PROGRAM Vision_Calibration
VAR
	
	Always_ON					:	BOOL	:=TRUE;	//상시ON
	Always_OFF					:	BOOL	:=FALSE;//상시OFF
	
	GVL_Calibration_Step: BOOL;
	TON_0: TON;
	TON_1: TON;
	TON_2: TON;
END_VAR
VAR // added by the converter: edge detectors and wires of the graphical bodies
    _w1 : BOOL;
END_VAR

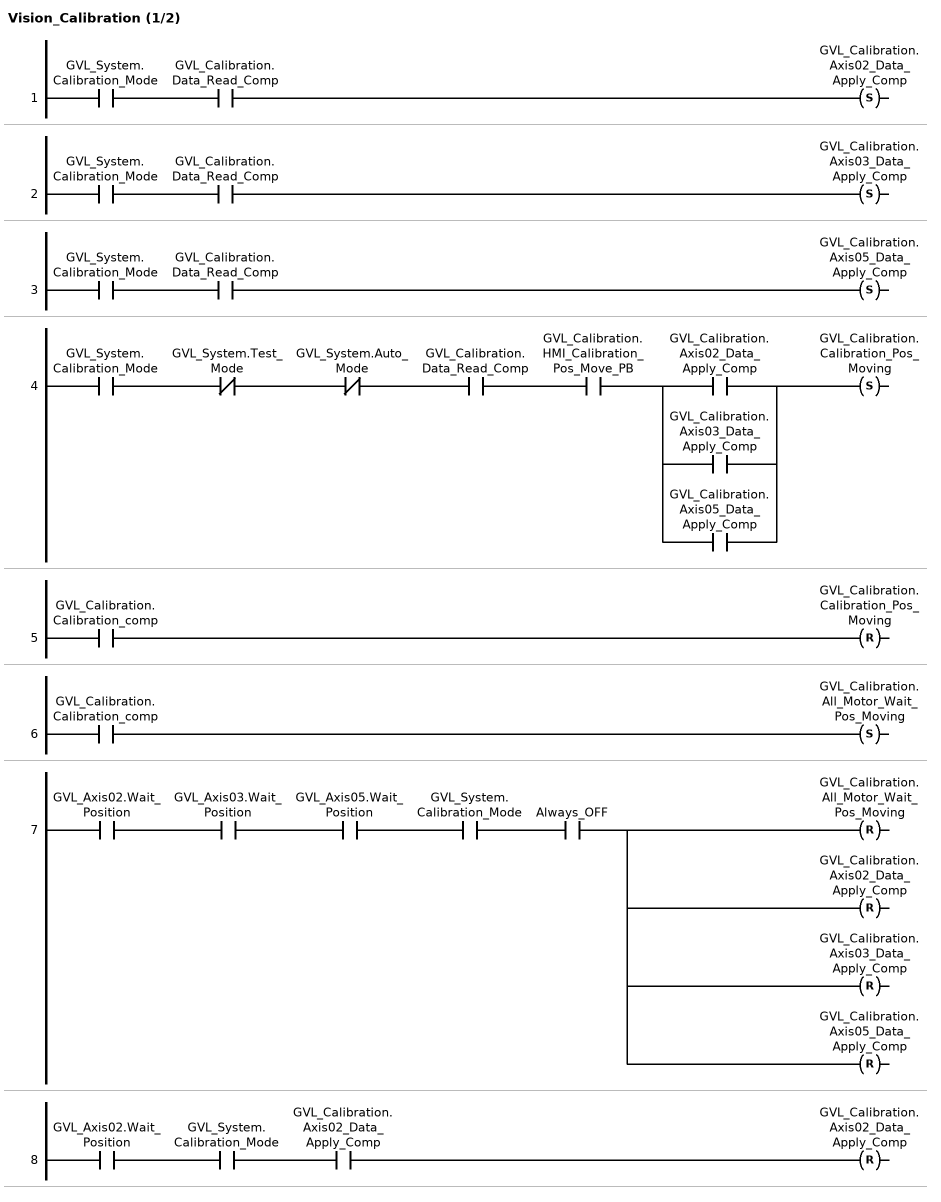
// NETWORK 1
GVL_Calibration.Axis02_Data_Apply_Comp S= GVL_System.Calibration_Mode AND GVL_Calibration.Data_Read_Comp;

// NETWORK 2
GVL_Calibration.Axis03_Data_Apply_Comp S= GVL_System.Calibration_Mode AND GVL_Calibration.Data_Read_Comp;

// NETWORK 3
GVL_Calibration.Axis05_Data_Apply_Comp S= GVL_System.Calibration_Mode AND GVL_Calibration.Data_Read_Comp;

// NETWORK 4
GVL_Calibration.Calibration_Pos_Moving S= GVL_System.Calibration_Mode AND NOT GVL_System.Test_Mode AND NOT GVL_System.Auto_Mode AND GVL_Calibration.Data_Read_Comp AND GVL_Calibration.HMI_Calibration_Pos_Move_PB AND (GVL_Calibration.Axis02_Data_Apply_Comp OR GVL_Calibration.Axis03_Data_Apply_Comp OR GVL_Calibration.Axis05_Data_Apply_Comp);

// NETWORK 5
GVL_Calibration.Calibration_Pos_Moving R= GVL_Calibration.Calibration_comp;

// NETWORK 6
GVL_Calibration.All_Motor_Wait_Pos_Moving S= GVL_Calibration.Calibration_comp;

// NETWORK 7
_w1 := GVL_Axis02.Wait_Position AND GVL_Axis03.Wait_Position AND GVL_Axis05.Wait_Position AND GVL_System.Calibration_Mode AND Always_OFF;
GVL_Calibration.All_Motor_Wait_Pos_Moving R= _w1;
GVL_Calibration.Axis02_Data_Apply_Comp R= _w1;
GVL_Calibration.Axis03_Data_Apply_Comp R= _w1;
GVL_Calibration.Axis05_Data_Apply_Comp R= _w1;

// NETWORK 8
GVL_Calibration.Axis02_Data_Apply_Comp R= GVL_Axis02.Wait_Position AND GVL_System.Calibration_Mode AND GVL_Calibration.Axis02_Data_Apply_Comp;

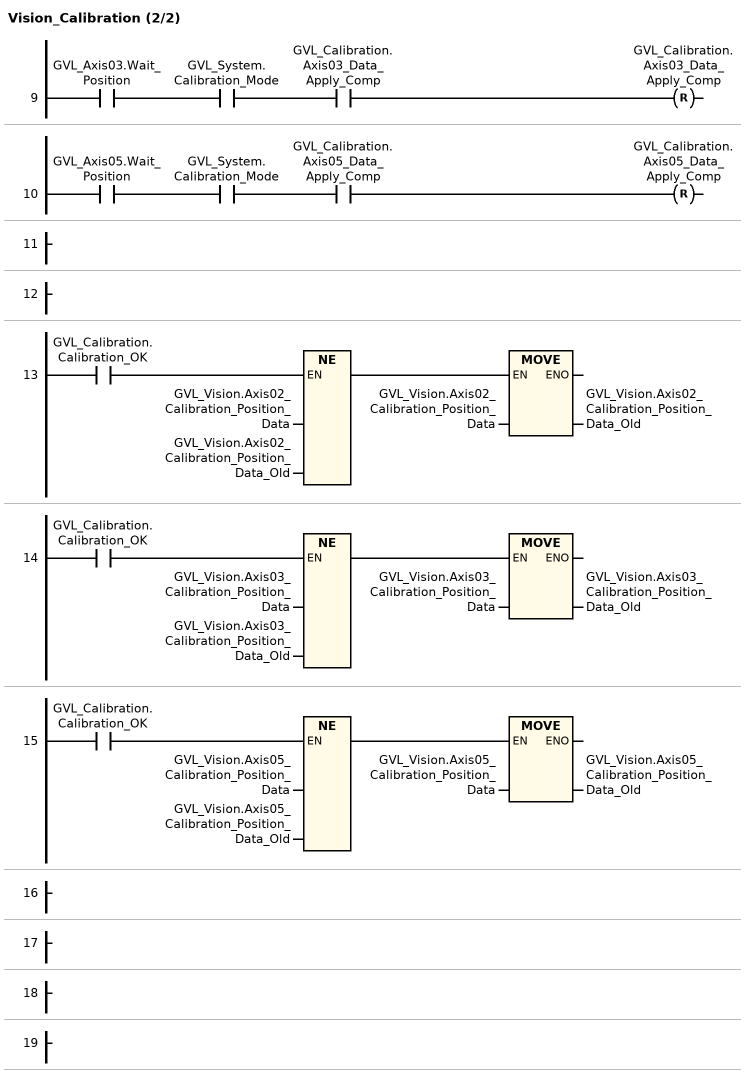
// NETWORK 9
GVL_Calibration.Axis03_Data_Apply_Comp R= GVL_Axis03.Wait_Position AND GVL_System.Calibration_Mode AND GVL_Calibration.Axis03_Data_Apply_Comp;

// NETWORK 10
GVL_Calibration.Axis05_Data_Apply_Comp R= GVL_Axis05.Wait_Position AND GVL_System.Calibration_Mode AND GVL_Calibration.Axis05_Data_Apply_Comp;

// NETWORK 11

// NETWORK 12

// NETWORK 13
IF GVL_Calibration.Calibration_OK AND GVL_Vision.Axis02_Calibration_Position_Data <> GVL_Vision.Axis02_Calibration_Position_Data_Old THEN
    GVL_Vision.Axis02_Calibration_Position_Data_Old := GVL_Vision.Axis02_Calibration_Position_Data;
END_IF

// NETWORK 14
IF GVL_Calibration.Calibration_OK AND GVL_Vision.Axis03_Calibration_Position_Data <> GVL_Vision.Axis03_Calibration_Position_Data_Old THEN
    GVL_Vision.Axis03_Calibration_Position_Data_Old := GVL_Vision.Axis03_Calibration_Position_Data;
END_IF

// NETWORK 15
IF GVL_Calibration.Calibration_OK AND GVL_Vision.Axis05_Calibration_Position_Data <> GVL_Vision.Axis05_Calibration_Position_Data_Old THEN
    GVL_Vision.Axis05_Calibration_Position_Data_Old := GVL_Vision.Axis05_Calibration_Position_Data;
END_IF

// NETWORK 16

// NETWORK 17

// NETWORK 18

// NETWORK 19

END_PROGRAM

(* stored: Version 1.1.0.1, ProductVersion 3.1.4024.15
   POU Vision_Calibration: Id {cb4ac576-599e-4820-9182-05726bb38b7c}, SpecialFunc None *)
